FUNCTION ASCF_CL_108_IF9 : Word
VAR_OUTPUT
	Out						: ASCF_UnionType;				//Result of the computation (Type: VDWord)
END_VAR

VAR_IN_OUT
	Arguments				: ARRAY[0..3] OF ASCF_UnionType;	//Arguments for the function (Argument[0]: VDWord, Argument[1]: VDWord, Argument[2]: VDWord, Argument[3]: VDWord)
END_VAR

VAR
	State1					: DWORD;
	BitMask					: DWORD;
	Command					: DWORD;
	PrevCommand				: DWORD;
	tempQCs					: ARRAY[0..3] OF BYTE;
	constDefaultUnionType	: ASCF_UnionType;				//Union type that holds only one of its possible data types at a time. The type can be selected via the "Typeselector". Independent of the selected type, every value has a quality code "VQC".
	constUnionTypes			: ASCF_EnumUnionTypes;			//Enumeration type of the valid values for the "Typeselector" of a "GVR_unionType"-UDT.
	constQualityCodes		: ASCF_QualityCodes;				//This enum encodes the defines quality codes for the MTP standard. The values are shown in HEX. The lowest value (1) has the highest priority.    | QC Name              | Value | Priority ||----------------------|:-----:|:--------:|| Failure              | 16#00 |    1     || Function Check       | 16#60 |    2     || Ma: INTenance Request  | 16#A4 |    3     || Out of Specification | 16#68 |    4     || OK                   | 16#80 |    5     || Out of Service       | 16#1C |    6     || No Status            | 16#FF |    7     |
	constErrors				: ASCF_CL_EnumErrors;				//Enumeration type of the error codes of the Adaptive Logic.
END_VAR



//#################################################################################################
{region "INITIALIZE VARIABLES"}
    Out := constDefaultUnionType;
{endregion}

//#################################################################################################
{region "PROCESS ARGUMENTS"}
    //-------------------------------------------------------------------------------------
    // State 1
    IF Arguments[0].Typeselector <> constUnionTypes.VDWord THEN
        ASCF_CL_108_IF9 := constErrors.InvalidType;
        RETURN;
    END_IF;
    
    //-------------------------------------------------------------------------------------
    // State 2
    IF Arguments[1].Typeselector <> constUnionTypes.VDWord THEN
        ASCF_CL_108_IF9 := constErrors.InvalidType;
        RETURN;
    END_IF;
    
    //-------------------------------------------------------------------------------------
    // Command
    IF Arguments[2].Typeselector <> constUnionTypes.VDWord THEN
        ASCF_CL_108_IF9 := constErrors.InvalidType;
        RETURN;
    END_IF;
    
    //-------------------------------------------------------------------------------------
    // Previous Command
    IF Arguments[3].Typeselector <> constUnionTypes.VDWord THEN
        ASCF_CL_108_IF9 := constErrors.InvalidType;
        RETURN;
    END_IF;
    
    State1 := Arguments[0].VDWord;
    BitMask := Arguments[1].VDWord;
    Command := Arguments[2].VDWord;
    PrevCommand := Arguments[3].VDWord;
    tempQCs[0] := Arguments[0].VQC;
    tempQCs[1] := Arguments[1].VQC;
    tempQCs[2] := Arguments[2].VQC;
    tempQCs[3] := Arguments[3].VQC;
{endregion}

//#################################################################################################
{region "OUTPUT"}
    Out.VQC := ASCF_CalcWQC(QC1 := ASCF_CalcWQC(QC1 := tempQCs[0], QC2 := tempQCs[1]), QC2 := ASCF_CalcWQC(QC1 := tempQCs[2], QC2 := tempQCs[3]));
    Out.Typeselector := constUnionTypes.VDWord;
    
    IF (State1 AND BitMask) <> 0 THEN
        Out.VDWord := Command;
    ELSE
        Out.VDWord := PrevCommand;
    END_IF;
    
    ASCF_CL_108_IF9 := constErrors.None;
{endregion}

END_FUNCTION

(* stored: Version 1.1.0.1, ProductVersion 3.1.4026.4
   POU ASCF_CL_108_IF9: Id {e128b763-1f5c-48ba-9038-ee94fa0608e3}, SpecialFunc None *)
